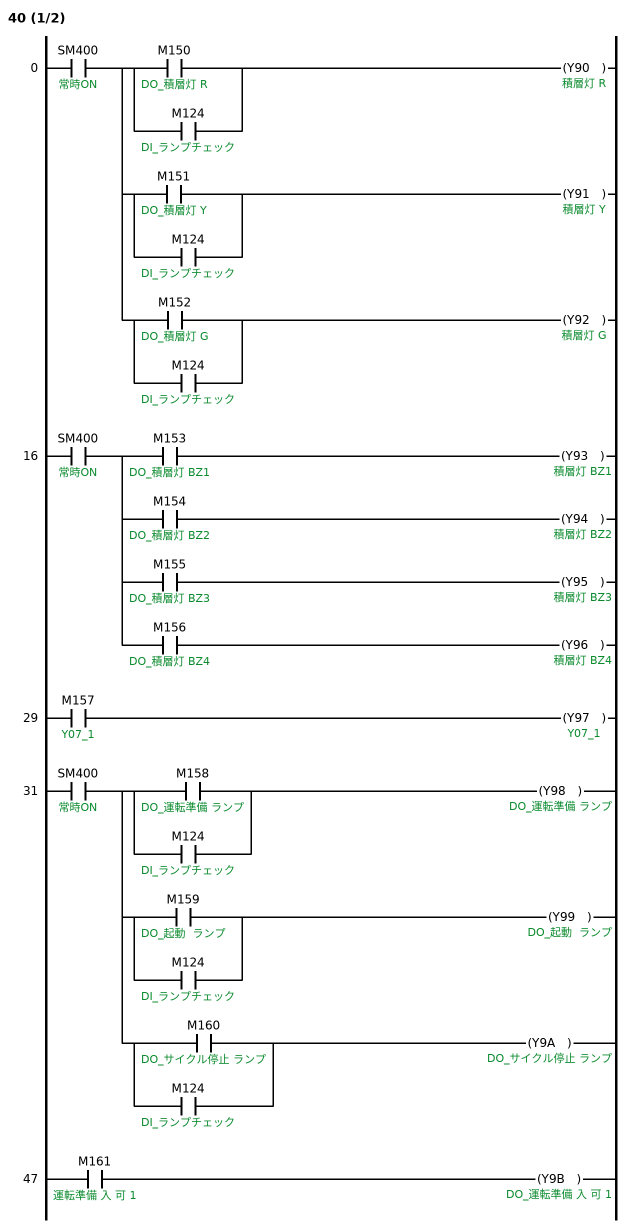
0     LD      SM400  ; 常時ON
      MPS
      LD      M150  ; DO_積層灯 R
      OR      M124  ; DI_ランプチェック
      ANB
      OUT     Y90  ; 積層灯 R
      MRD
      LD      M151  ; DO_積層灯 Y
      OR      M124  ; DI_ランプチェック
      ANB
      OUT     Y91  ; 積層灯 Y
      MPP
      LD      M152  ; DO_積層灯 G
      OR      M124  ; DI_ランプチェック
      ANB
      OUT     Y92  ; 積層灯 G
16    LD      SM400  ; 常時ON
      MPS
      AND     M153  ; DO_積層灯 BZ1
      OUT     Y93  ; 積層灯 BZ1
      MRD
      AND     M154  ; DO_積層灯 BZ2
      OUT     Y94  ; 積層灯 BZ2
      MRD
      AND     M155  ; DO_積層灯 BZ3
      OUT     Y95  ; 積層灯 BZ3
      MPP
      AND     M156  ; DO_積層灯 BZ4
      OUT     Y96  ; 積層灯 BZ4
29    LD      M157  ; Y07_1
      OUT     Y97  ; Y07_1
31    LD      SM400  ; 常時ON
      MPS
      LD      M158  ; DO_運転準備 ランプ
      OR      M124  ; DI_ランプチェック
      ANB
      OUT     Y98  ; DO_運転準備 ランプ
      MRD
      LD      M159  ; DO_起動  ランプ
      OR      M124  ; DI_ランプチェック
      ANB
      OUT     Y99  ; DO_起動  ランプ
      MPP
      LD      M160  ; DO_サイクル停止 ランプ
      OR      M124  ; DI_ランプチェック
      ANB
      OUT     Y9A  ; DO_サイクル停止 ランプ
47    LD      M161  ; 運転準備 入 可 1
      OUT     Y9B  ; DO_運転準備 入 可 1
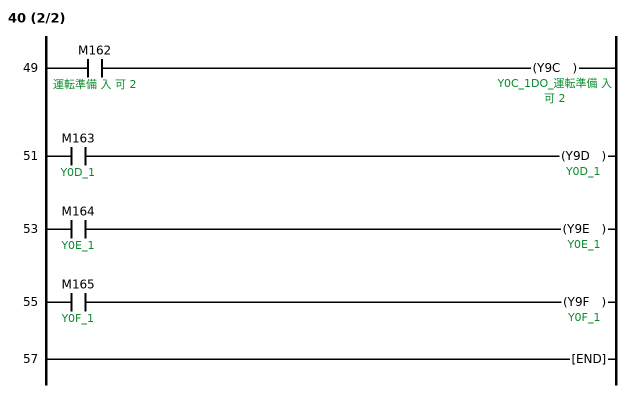
49    LD      M162  ; 運転準備 入 可 2
      OUT     Y9C  ; Y0C_1DO_運転準備 入 可 2
51    LD      M163  ; Y0D_1
      OUT     Y9D  ; Y0D_1
53    LD      M164  ; Y0E_1
      OUT     Y9E  ; Y0E_1
55    LD      M165  ; Y0F_1
      OUT     Y9F  ; Y0F_1
57    END
END_PROGRAM

PROGRAM 42  // スタッカー 出力
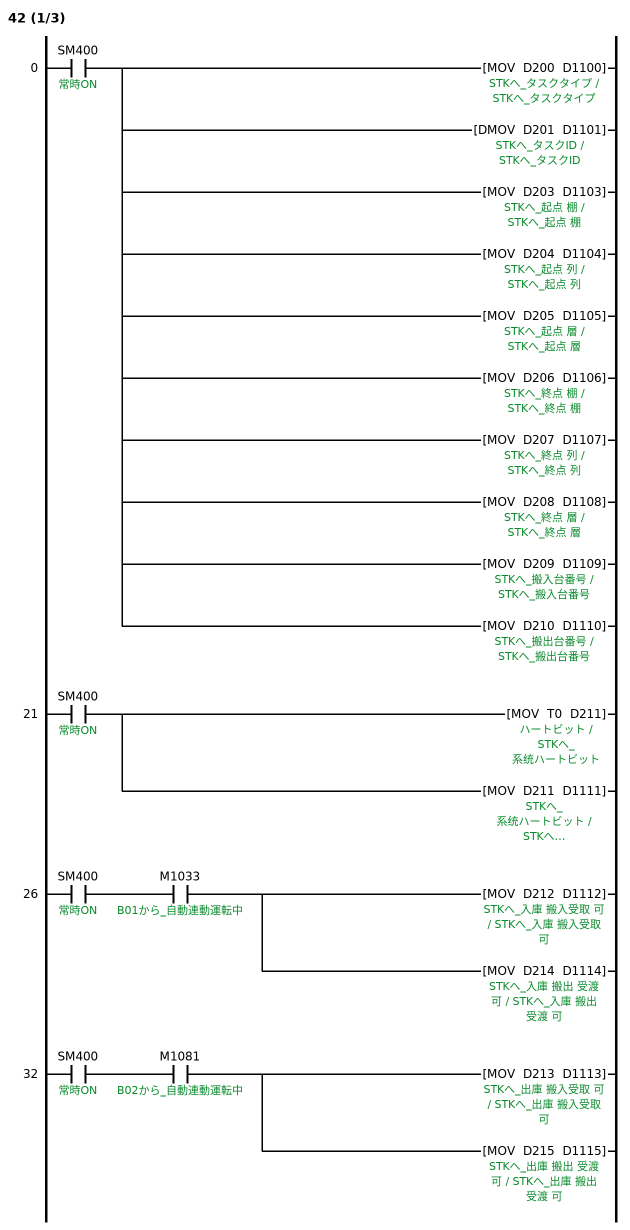
0     LD      SM400  ; 常時ON
      MOV     D200 D1100  ; STKへ_タスクタイプ / STKへ_タスクタイプ
      DMOV    D201 D1101  ; STKへ_タスクID / STKへ_タスクID
      MOV     D203 D1103  ; STKへ_起点 棚 / STKへ_起点 棚
      MOV     D204 D1104  ; STKへ_起点 列 / STKへ_起点 列
      MOV     D205 D1105  ; STKへ_起点 層 / STKへ_起点 層
      MOV     D206 D1106  ; STKへ_終点 棚 / STKへ_終点 棚
      MOV     D207 D1107  ; STKへ_終点 列 / STKへ_終点 列
      MOV     D208 D1108  ; STKへ_終点 層 / STKへ_終点 層
      MOV     D209 D1109  ; STKへ_搬入台番号 / STKへ_搬入台番号
      MOV     D210 D1110  ; STKへ_搬出台番号 / STKへ_搬出台番号
21    LD      SM400  ; 常時ON
      MOV     T0 D211  ; ハートビット / STKへ_系统ハートビット
      MOV     D211 D1111  ; STKへ_系统ハートビット
26    LD      SM400  ; 常時ON
      AND     M1033  ; B01から_自動連動運転中
      MOV     D212 D1112  ; STKへ_入庫 搬入受取 可 / STKへ_入庫 搬入受取 可
      MOV     D214 D1114  ; STKへ_入庫 搬出 受渡 可 / STKへ_入庫 搬出 受渡 可
32    LD      SM400  ; 常時ON
      AND     M1081  ; B02から_自動連動運転中
      MOV     D213 D1113  ; STKへ_出庫 搬入受取 可 / STKへ_出庫 搬入受取 可
      MOV     D215 D1115  ; STKへ_出庫 搬出 受渡 可 / STKへ_出庫 搬出 受渡 可
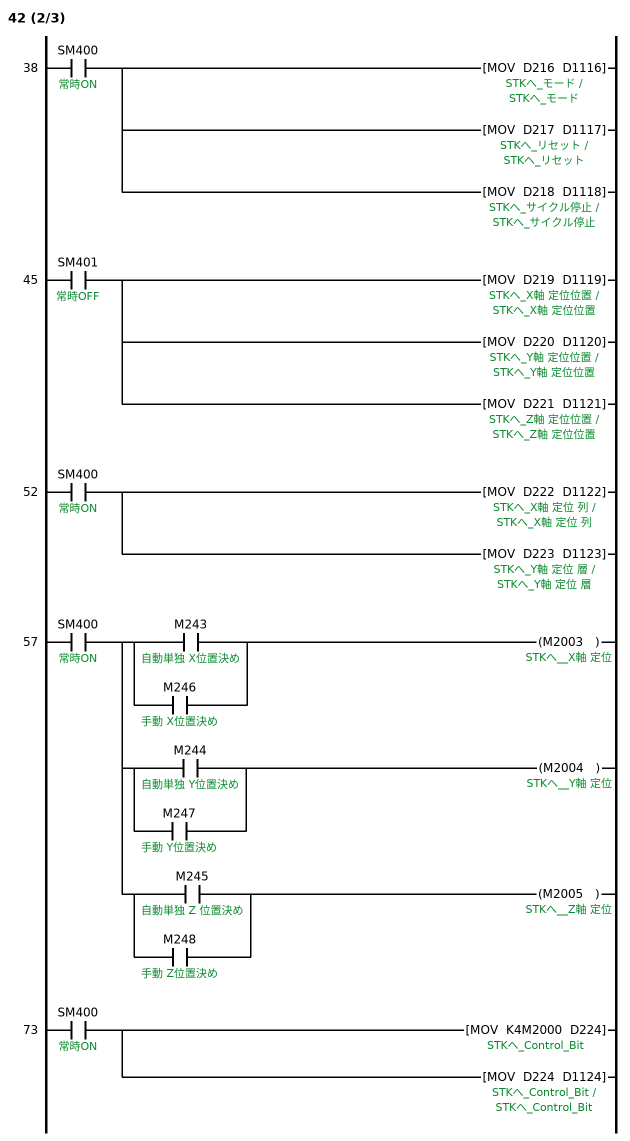
38    LD      SM400  ; 常時ON
      MOV     D216 D1116  ; STKへ_モード / STKへ_モード
      MOV     D217 D1117  ; STKへ_リセット / STKへ_リセット
      MOV     D218 D1118  ; STKへ_サイクル停止 / STKへ_サイクル停止
45    LD      SM401  ; 常時OFF
      MOV     D219 D1119  ; STKへ_X軸 定位位置 / STKへ_X軸 定位位置
      MOV     D220 D1120  ; STKへ_Y軸 定位位置 / STKへ_Y軸 定位位置
      MOV     D221 D1121  ; STKへ_Z軸 定位位置 / STKへ_Z軸 定位位置
52    LD      SM400  ; 常時ON
      MOV     D222 D1122  ; STKへ_X軸 定位 列 / STKへ_X軸 定位 列
      MOV     D223 D1123  ; STKへ_Y軸 定位 層 / STKへ_Y軸 定位 層
57    LD      SM400  ; 常時ON
      MPS
      LD      M243  ; 自動単独 X位置決め
      OR      M246  ; 手動 X位置決め
      ANB
      OUT     M2003  ; STKへ__X軸 定位
      MRD
      LD      M244  ; 自動単独 Y位置決め
      OR      M247  ; 手動 Y位置決め
      ANB
      OUT     M2004  ; STKへ__Y軸 定位
      MPP
      LD      M245  ; 自動単独 Z 位置決め
      OR      M248  ; 手動 Z位置決め
      ANB
      OUT     M2005  ; STKへ__Z軸 定位
73    LD      SM400  ; 常時ON
      MOV     K4M2000 D224  ; STKへ_手動制御リクエスト / STKへ_Control_Bit
      MOV     D224 D1124  ; STKへ_Control_Bit
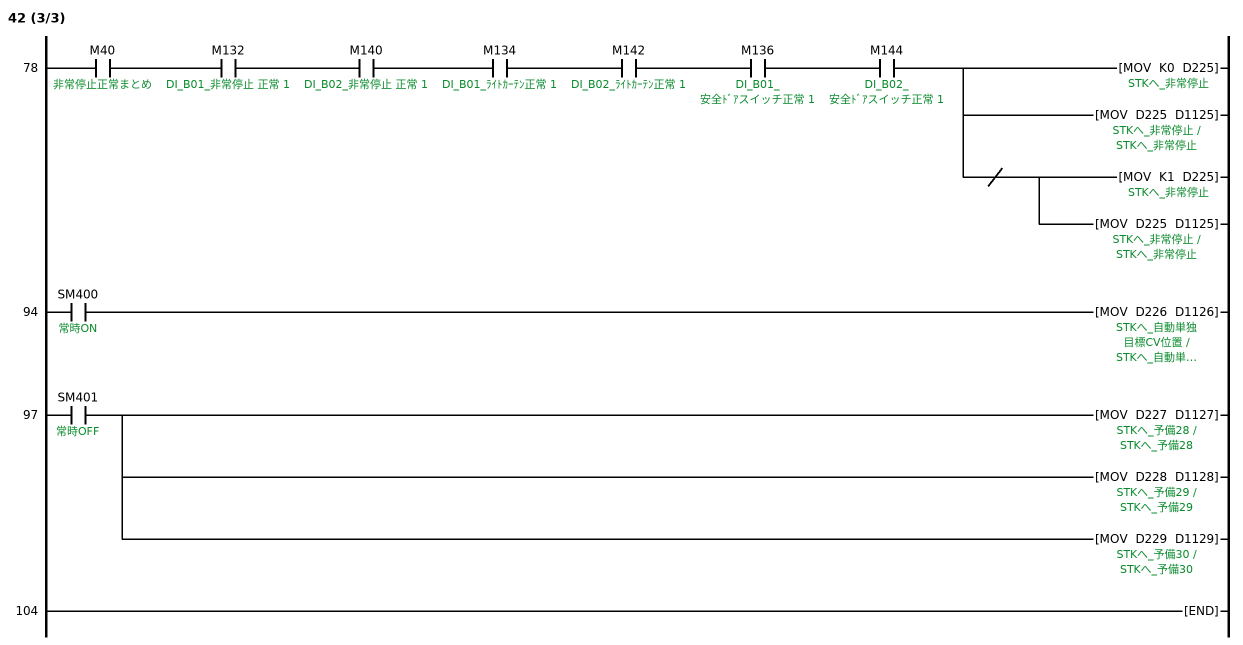
78    LD      M40  ; 非常停止正常まとめ
      AND     M132  ; DI_B01_非常停止 正常 1
      AND     M140  ; DI_B02_非常停止 正常 1
      AND     M134  ; DI_B01_ﾗｲﾄｶｰﾃﾝ正常 1
      AND     M142  ; DI_B02_ﾗｲﾄｶｰﾃﾝ正常 1
      AND     M136  ; DI_B01_安全ﾄﾞｱスイッチ正常 1
      AND     M144  ; DI_B02_安全ﾄﾞｱスイッチ正常 1
      MOV     K0 D225  ; STKへ_非常停止
      MOV     D225 D1125  ; STKへ_非常停止
      INV
      MOV     K1 D225
      MOV     D225 D1125
94    LD      SM400  ; 常時ON
      MOV     D226 D1126  ; STKへ_自動単独 目標CV位置 / STKへ_自動単独 目標CV位置
97    LD      SM401  ; 常時OFF
      MOV     D227 D1127  ; STKへ_予備28 / STKへ_予備28
      MOV     D228 D1128  ; STKへ_予備29 / STKへ_予備29
      MOV     D229 D1129  ; STKへ_予備30 / STKへ_予備30
104   END
END_PROGRAM

PROGRAM 43  // WMS 出力
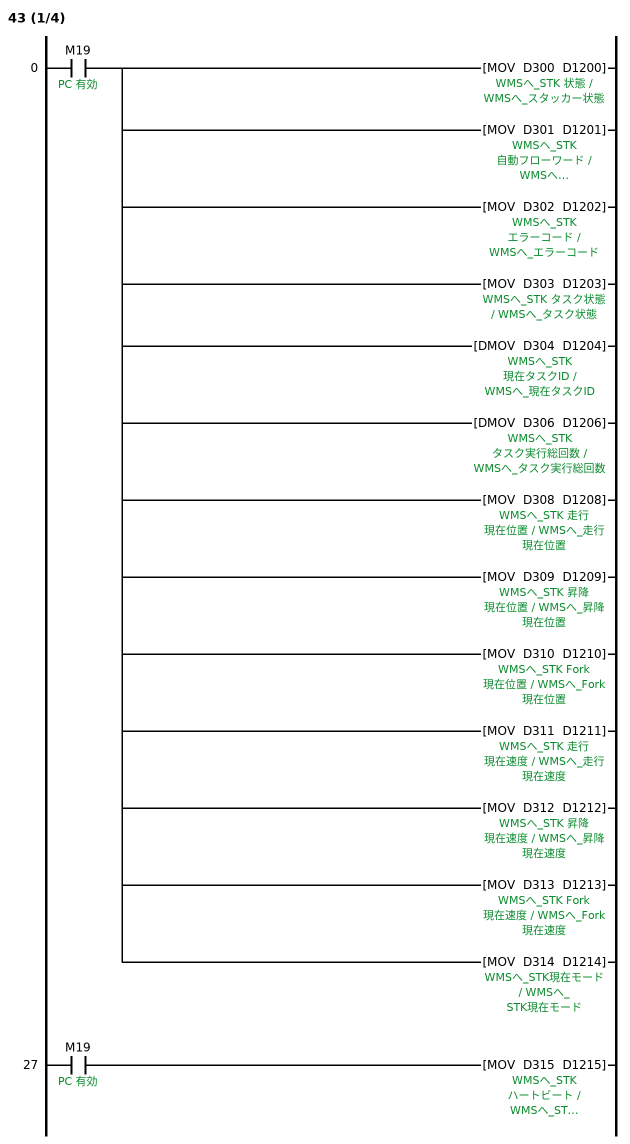
0     LD      M19  ; PC 有効
      MOV     D300 D1200  ; WMSへ_STK 状態 / WMSへ_スタッカー状態
      MOV     D301 D1201  ; WMSへ_STK 自動フローワード / WMSへ_自動フローワード
      MOV     D302 D1202  ; WMSへ_STK エラーコード / WMSへ_エラーコード
      MOV     D303 D1203  ; WMSへ_STK タスク状態 / WMSへ_タスク状態
      DMOV    D304 D1204  ; WMSへ_STK 現在タスクID / WMSへ_現在タスクID
      DMOV    D306 D1206  ; WMSへ_STK タスク実行総回数 / WMSへ_タスク実行総回数
      MOV     D308 D1208  ; WMSへ_STK 走行 現在位置 / WMSへ_走行 現在位置
      MOV     D309 D1209  ; WMSへ_STK 昇降 現在位置 / WMSへ_昇降 現在位置
      MOV     D310 D1210  ; WMSへ_STK Fork 現在位置 / WMSへ_Fork 現在位置
      MOV     D311 D1211  ; WMSへ_STK 走行 現在速度 / WMSへ_走行 現在速度
      MOV     D312 D1212  ; WMSへ_STK 昇降 現在速度 / WMSへ_昇降 現在速度
      MOV     D313 D1213  ; WMSへ_STK Fork 現在速度 / WMSへ_Fork 現在速度
      MOV     D314 D1214  ; WMSへ_STK現在モード / WMSへ_STK現在モード
27    LD      M19  ; PC 有効
      MOV     D315 D1215  ; WMSへ_STK ハートビート / WMSへ_STK ハートビート
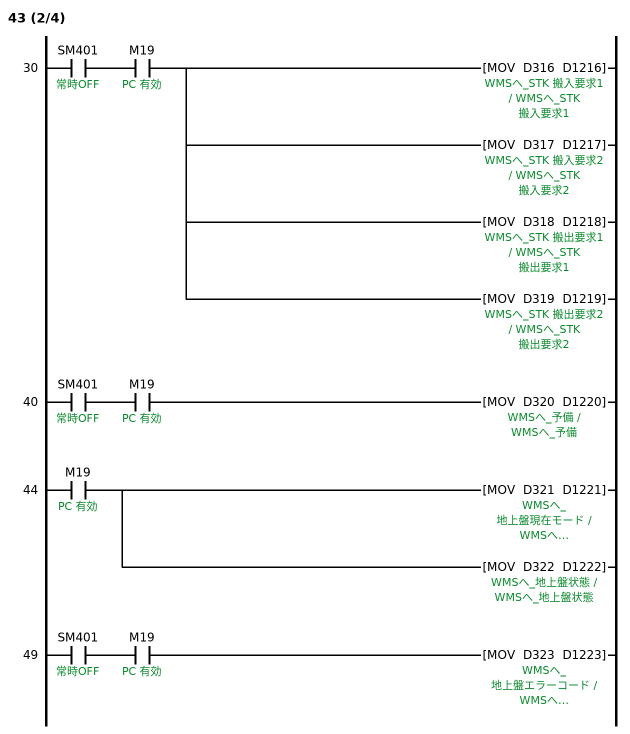
30    LD      SM401  ; 常時OFF
      AND     M19  ; PC 有効
      MOV     D316 D1216  ; WMSへ_STK 搬入要求1 / WMSへ_STK 搬入要求1
      MOV     D317 D1217  ; WMSへ_STK 搬入要求2 / WMSへ_STK 搬入要求2
      MOV     D318 D1218  ; WMSへ_STK 搬出要求1 / WMSへ_STK 搬出要求1
      MOV     D319 D1219  ; WMSへ_STK 搬出要求2 / WMSへ_STK 搬出要求2
40    LD      SM401  ; 常時OFF
      AND     M19  ; PC 有効
      MOV     D320 D1220  ; WMSへ_予備 / WMSへ_予備
44    LD      M19  ; PC 有効
      MOV     D321 D1221  ; WMSへ_地上盤現在モード / WMSへ_地上盤現在モード
      MOV     D322 D1222  ; WMSへ_地上盤状態 / WMSへ_地上盤状態
49    LD      SM401  ; 常時OFF
      AND     M19  ; PC 有効
      MOV     D323 D1223  ; WMSへ_地上盤エラーコード / WMSへ_地上盤エラーコード
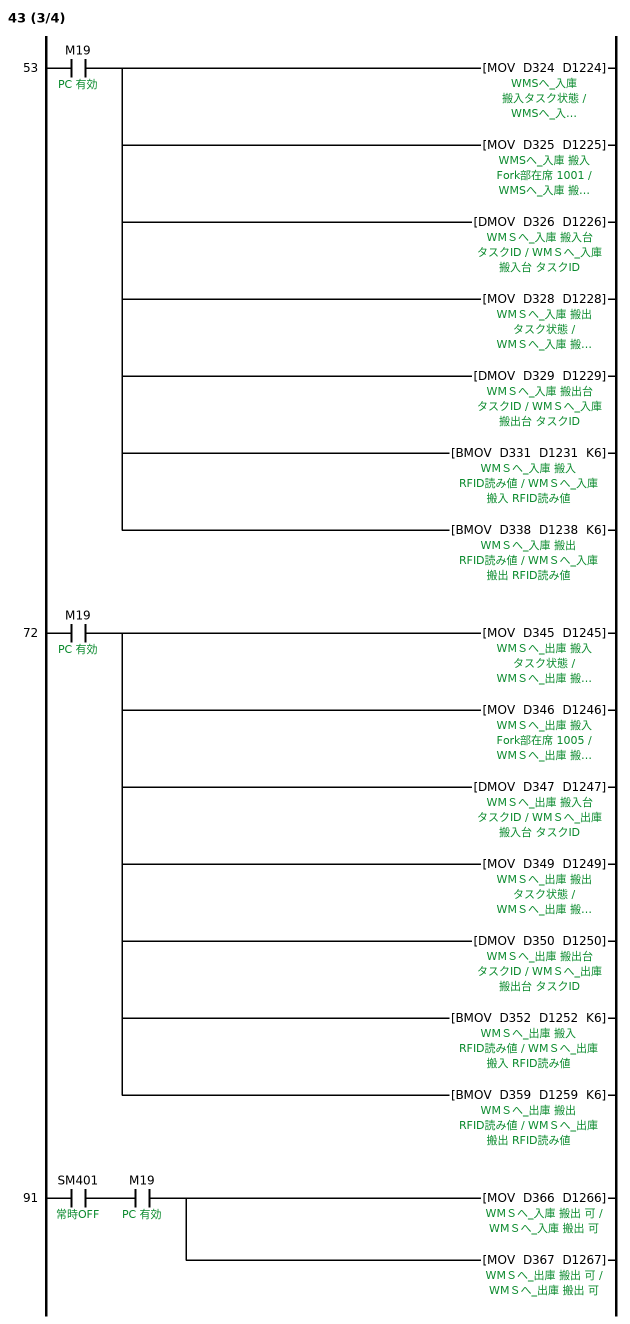
53    LD      M19  ; PC 有効
      MOV     D324 D1224  ; WMSへ_入庫 搬入タスク状態 / WMSへ_入庫 搬入タスク状態
      MOV     D325 D1225  ; WMSへ_入庫 搬入 Fork部在席 1001 / WMSへ_入庫 搬入 Fork在席
      DMOV    D326 D1226  ; WMＳへ_入庫 搬入台 タスクID / WMＳへ_入庫 搬入台 タスクID
      MOV     D328 D1228  ; WMＳへ_入庫 搬出 タスク状態 / WMＳへ_入庫 搬出 タスク状態
      DMOV    D329 D1229  ; WMＳへ_入庫 搬出台 タスクID / WMＳへ_入庫 搬出台 タスクID
      BMOV    D331 D1231 K6  ; WMＳへ_入庫 搬入 RFID読み値 / WMＳへ_入庫 搬入 RFID読み値
      BMOV    D338 D1238 K6  ; WMＳへ_入庫 搬出 RFID読み値 / WMＳへ_入庫 搬出 RFID読み値
72    LD      M19  ; PC 有効
      MOV     D345 D1245  ; WMＳへ_出庫 搬入 タスク状態 / WMＳへ_出庫 搬入 タスク状態
      MOV     D346 D1246  ; WMＳへ_出庫 搬入 Fork部在席 1005 / WMＳへ_出庫 搬入 Fork部在席
      DMOV    D347 D1247  ; WMＳへ_出庫 搬入台 タスクID / WMＳへ_出庫 搬入台 タスクID
      MOV     D349 D1249  ; WMＳへ_出庫 搬出 タスク状態 / WMＳへ_出庫 搬出 タスク状態
      DMOV    D350 D1250  ; WMＳへ_出庫 搬出台 タスクID / WMＳへ_出庫 搬出台 タスクID
      BMOV    D352 D1252 K6  ; WMＳへ_出庫 搬入 RFID読み値 / WMＳへ_出庫 搬入 RFID読み値
      BMOV    D359 D1259 K6  ; WMＳへ_出庫 搬出 RFID読み値 / WMＳへ_出庫 搬出 RFID読み値
91    LD      SM401  ; 常時OFF
      AND     M19  ; PC 有効
      MOV     D366 D1266  ; WMＳへ_入庫 搬出 可 / WMＳへ_入庫 搬出 可
      MOV     D367 D1267  ; WMＳへ_出庫 搬出 可 / WMＳへ_出庫 搬出 可
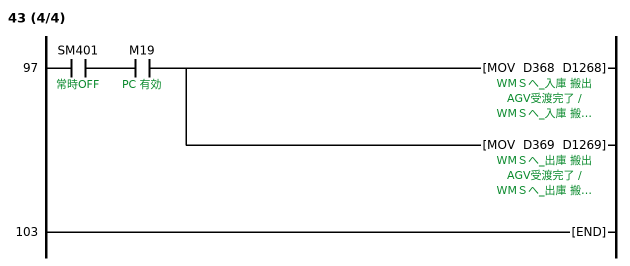
97    LD      SM401  ; 常時OFF
      AND     M19  ; PC 有効
      MOV     D368 D1268  ; WMＳへ_入庫 搬出 AGV受渡完了 / WMＳへ_入庫 搬出 AGV受渡完了
      MOV     D369 D1269  ; WMＳへ_出庫 搬出 AGV受渡完了 / WMＳへ_出庫 搬出 AGV受渡完了
103   END
END_PROGRAM

FUNCTION_BLOCK I+ST_02f34114d45741f9
VAR_INPUT
  __IST_EN_IN : BOOL;
END_VAR
VAR_OUTPUT
  __IST_EN_OUT : BOOL;
END_VAR
(* IST HEADER START *)
IF NOT __IST_EN_IN THEN __IST_EN_OUT:=FALSE; RETURN; END_IF;
(* VERSION=1:TYPE=STB *)
(* IST HEADER END *)
Z0:=(Alone.起点列 - 1) * 5 + (Alone.起点層 - 1); (*起点位置*)
END_FUNCTION_BLOCK

FUNCTION_BLOCK I+ST_08ba2391820a4452
VAR_INPUT
  __IST_EN_IN : BOOL;
END_VAR
VAR_OUTPUT
  __IST_EN_OUT : BOOL;
END_VAR
(* IST HEADER START *)
IF NOT __IST_EN_IN THEN __IST_EN_OUT:=FALSE; RETURN; END_IF;
(* VERSION=1:TYPE=STB *)
(* IST HEADER END *)
Z1:=(Alone.終点列 - 1) * 5 + (Alone.終点層 - 1); (*目的位置*)
END_FUNCTION_BLOCK

PROGRAM 13  // STK 自動/単独ﾓｰﾄﾞ
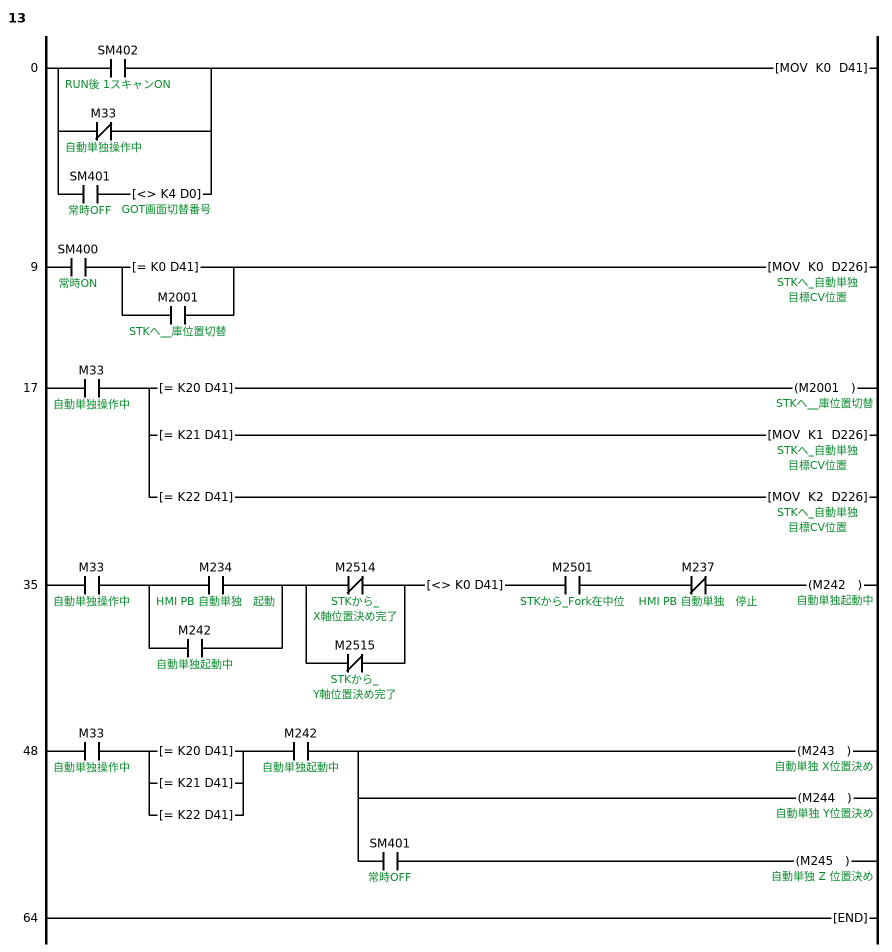
0     LD      SM402  ; RUN後 1スキャンON
      ORI     M33  ; 自動単独操作中
      LD      SM401  ; 常時OFF
      AND<>   K4 D0  ; GOT画面切替番号
      ORB
      MOV     K0 D41
9     LD      SM400  ; 常時ON
      LD=     K0 D41
      OR      M2001  ; STKへ__庫位置切替
      ANB
      MOV     K0 D226  ; STKへ_自動単独 目標CV位置
17    LD      M33  ; 自動単独操作中
      MPS
      AND=    K20 D41
      OUT     M2001  ; STKへ__庫位置切替
      MRD
      AND=    K21 D41
      MOV     K1 D226
      MPP
      AND=    K22 D41
      MOV     K2 D226
35    LD      M33  ; 自動単独操作中
      LD      M234  ; HMI PB 自動単独　起動
      OR      M242  ; 自動単独起動中
      ANB
      LDI     M2514  ; STKから_X軸位置決め完了
      ORI     M2515  ; STKから_Y軸位置決め完了
      ANB
      AND<>   K0 D41
      AND     M2501  ; STKから_Fork在中位
      ANI     M237  ; HMI PB 自動単独　停止
      OUT     M242  ; 自動単独起動中
48    LD      M33  ; 自動単独操作中
      LD=     K20 D41
      OR=     K21 D41
      OR=     K22 D41
      ANB
      AND     M242  ; 自動単独起動中
      OUT     M243  ; 自動単独 X位置決め
      OUT     M244  ; 自動単独 Y位置決め
      AND     SM401  ; 常時OFF
      OUT     M245  ; 自動単独 Z 位置決め
64    END
END_PROGRAM

PROGRAM 04  // B01 CC-LinkIE XYD 入力
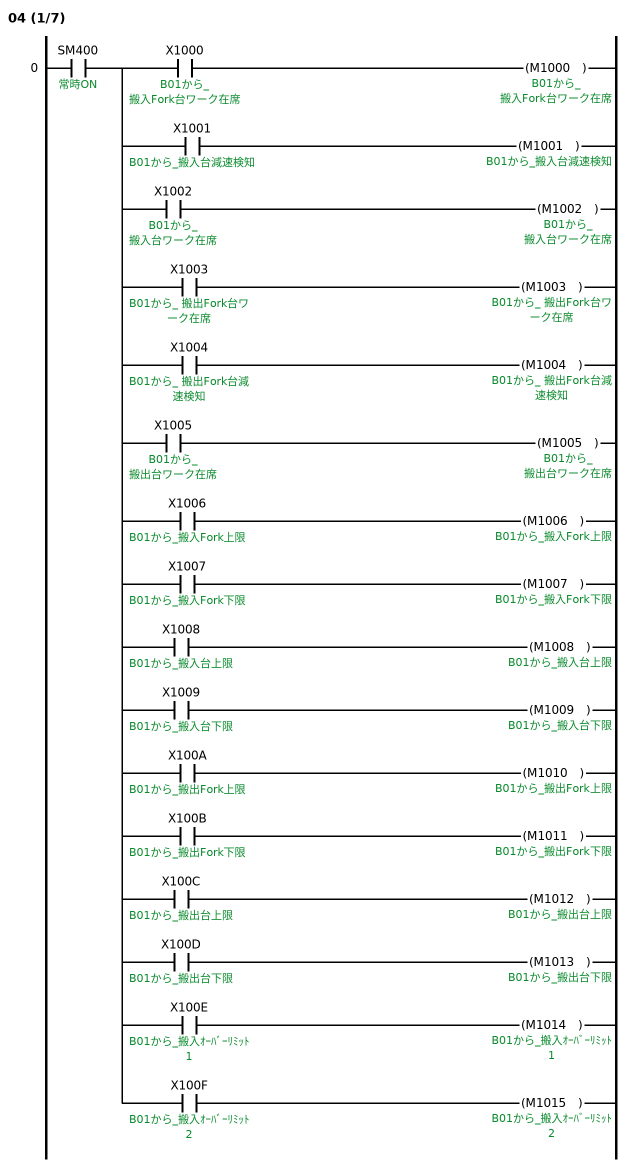
0     LD      SM400  ; 常時ON
      MPS
      AND     X1000  ; B01から_搬入Fork台ワーク在席
      OUT     M1000  ; B01から_搬入Fork台ワーク在席
      MRD
      AND     X1001  ; B01から_搬入台減速検知
      OUT     M1001  ; B01から_搬入台減速検知
      MRD
      AND     X1002  ; B01から_搬入台ワーク在席
      OUT     M1002  ; B01から_搬入台ワーク在席
      MRD
      AND     X1003  ; B01から_ 搬出Fork台ワーク在席
      OUT     M1003  ; B01から_ 搬出Fork台ワーク在席
      MRD
      AND     X1004  ; B01から_ 搬出Fork台減速検知
      OUT     M1004  ; B01から_ 搬出Fork台減速検知
      MRD
      AND     X1005  ; B01から_ 搬出台ワーク在席
      OUT     M1005  ; B01から_ 搬出台ワーク在席
      MRD
      AND     X1006  ; B01から_搬入Fork上限
      OUT     M1006  ; B01から_搬入Fork上限
      MRD
      AND     X1007  ; B01から_搬入Fork下限
      OUT     M1007  ; B01から_搬入Fork下限
      MRD
      AND     X1008  ; B01から_搬入台上限
      OUT     M1008  ; B01から_搬入台上限
      MRD
      AND     X1009  ; B01から_搬入台下限
      OUT     M1009  ; B01から_搬入台下限
      MRD
      AND     X100A  ; B01から_搬出Fork上限
      OUT     M1010  ; B01から_搬出Fork上限
      MRD
      AND     X100B  ; B01から_搬出Fork下限
      OUT     M1011  ; B01から_搬出Fork下限
      MRD
      AND     X100C  ; B01から_搬出台上限
      OUT     M1012  ; B01から_搬出台上限
      MRD
      AND     X100D  ; B01から_搬出台下限
      OUT     M1013  ; B01から_搬出台下限
      MRD
      AND     X100E  ; B01から_搬入ｵｰﾊﾞｰﾘﾐｯﾄ 1
      OUT     M1014  ; B01から_搬入ｵｰﾊﾞｰﾘﾐｯﾄ 1
      MPP
      AND     X100F  ; B01から_搬入ｵｰﾊﾞｰﾘﾐｯﾄ 2
      OUT     M1015  ; B01から_搬入ｵｰﾊﾞｰﾘﾐｯﾄ 2
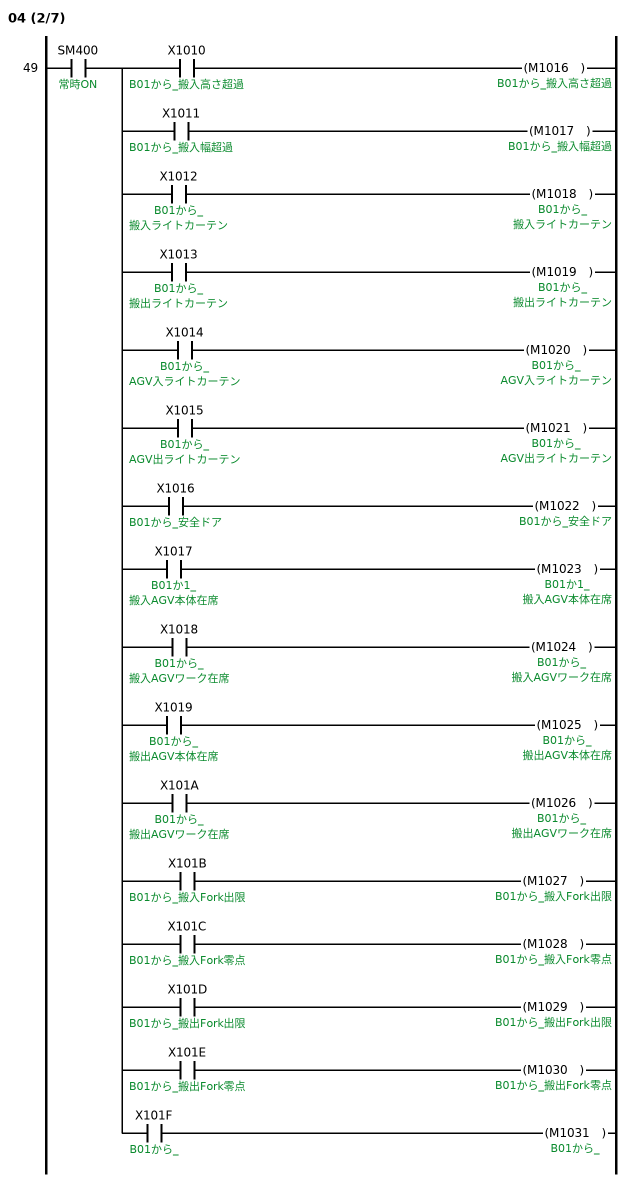
49    LD      SM400  ; 常時ON
      MPS
      AND     X1010  ; B01から_搬入高さ超過
      OUT     M1016  ; B01から_搬入高さ超過
      MRD
      AND     X1011  ; B01から_搬入幅超過
      OUT     M1017  ; B01から_搬入幅超過
      MRD
      AND     X1012  ; B01から_搬入ライトカーテン
      OUT     M1018  ; B01から_搬入ライトカーテン
      MRD
      AND     X1013  ; B01から_搬出ライトカーテン
      OUT     M1019  ; B01から_搬出ライトカーテン
      MRD
      AND     X1014  ; B01から_AGV入ライトカーテン
      OUT     M1020  ; B01から_AGV入ライトカーテン
      MRD
      AND     X1015  ; B01から_AGV出ライトカーテン
      OUT     M1021  ; B01から_AGV出ライトカーテン
      MRD
      AND     X1016  ; B01から_安全ドア
      OUT     M1022  ; B01から_安全ドア
      MRD
      AND     X1017  ; B01か1_搬入AGV本体在席
      OUT     M1023  ; B01か1_搬入AGV本体在席
      MRD
      AND     X1018  ; B01から_搬入AGVワーク在席
      OUT     M1024  ; B01から_搬入AGVワーク在席
      MRD
      AND     X1019  ; B01から_搬出AGV本体在席
      OUT     M1025  ; B01から_搬出AGV本体在席
      MRD
      AND     X101A  ; B01から_搬出AGVワーク在席
      OUT     M1026  ; B01から_搬出AGVワーク在席
      MRD
      AND     X101B  ; B01から_搬入Fork出限
      OUT     M1027  ; B01から_搬入Fork出限
      MRD
      AND     X101C  ; B01から_搬入Fork零点
      OUT     M1028  ; B01から_搬入Fork零点
      MRD
      AND     X101D  ; B01から_搬出Fork出限
      OUT     M1029  ; B01から_搬出Fork出限
      MRD
      AND     X101E  ; B01から_搬出Fork零点
      OUT     M1030  ; B01から_搬出Fork零点
      MPP
      AND     X101F  ; B01から_
      OUT     M1031  ; B01から_
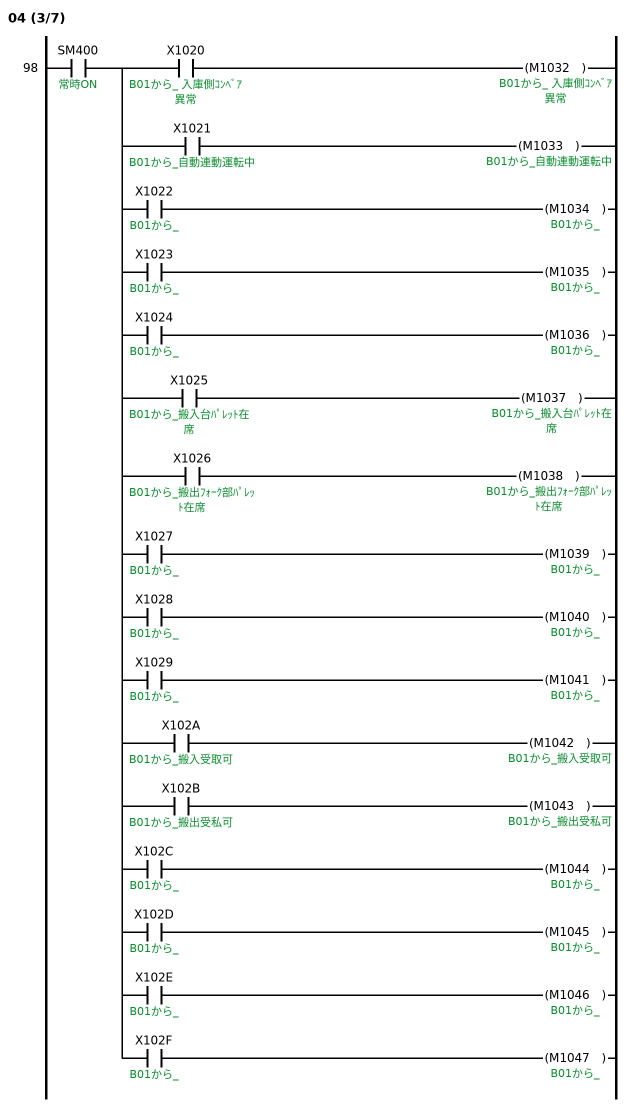
98    LD      SM400  ; 常時ON
      MPS
      AND     X1020  ; B01から_ 入庫側ｺﾝﾍﾞｱ 異常
      OUT     M1032  ; B01から_ 入庫側ｺﾝﾍﾞｱ 異常
      MRD
      AND     X1021  ; B01から_自動連動運転中
      OUT     M1033  ; B01から_自動連動運転中
      MRD
      AND     X1022  ; B01から_
      OUT     M1034  ; B01から_
      MRD
      AND     X1023  ; B01から_
      OUT     M1035  ; B01から_
      MRD
      AND     X1024  ; B01から_
      OUT     M1036  ; B01から_
      MRD
      AND     X1025  ; B01から_搬入台ﾊﾟﾚｯﾄ在席
      OUT     M1037  ; B01から_搬入台ﾊﾟﾚｯﾄ在席
      MRD
      AND     X1026  ; B01から_搬出ﾌｫｰｸ部ﾊﾟﾚｯﾄ在席
      OUT     M1038  ; B01から_搬出ﾌｫｰｸ部ﾊﾟﾚｯﾄ在席
      MRD
      AND     X1027  ; B01から_
      OUT     M1039  ; B01から_
      MRD
      AND     X1028  ; B01から_
      OUT     M1040  ; B01から_
      MRD
      AND     X1029  ; B01から_
      OUT     M1041  ; B01から_
      MRD
      AND     X102A  ; B01から_搬入受取可
      OUT     M1042  ; B01から_搬入受取可
      MRD
      AND     X102B  ; B01から_搬出受私可
      OUT     M1043  ; B01から_搬出受私可
      MRD
      AND     X102C  ; B01から_
      OUT     M1044  ; B01から_
      MRD
      AND     X102D  ; B01から_
      OUT     M1045  ; B01から_
      MRD
      AND     X102E  ; B01から_
      OUT     M1046  ; B01から_
      MPP
      AND     X102F  ; B01から_
      OUT     M1047  ; B01から_
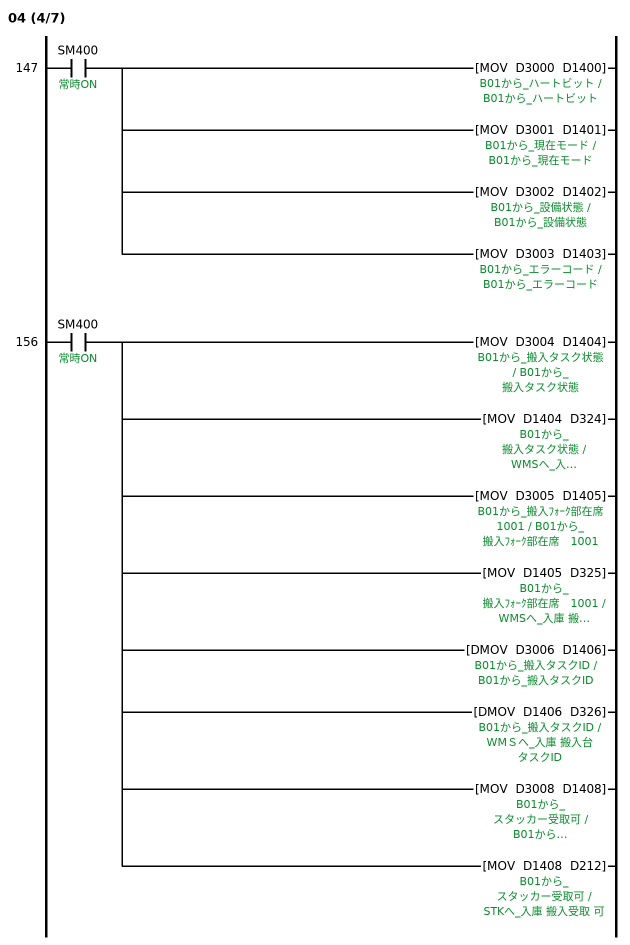
147   LD      SM400  ; 常時ON
      MOV     D3000 D1400  ; B01から_ハートビット / B01から_ハートビット
      MOV     D3001 D1401  ; B01から_現在モード / B01から_現在モード
      MOV     D3002 D1402  ; B01から_設備状態 / B01から_設備状態
      MOV     D3003 D1403  ; B01から_エラーコード / B01から_エラーコード
156   LD      SM400  ; 常時ON
      MOV     D3004 D1404  ; B01から_搬入タスク状態 / B01から_搬入タスク状態
      MOV     D1404 D324  ; WMSへ_入庫 搬入タスク状態
      MOV     D3005 D1405  ; B01から_搬入ﾌｫｰｸ部在席　1001 / B01から_搬入ﾌｫｰｸ部在席　1001
      MOV     D1405 D325  ; WMSへ_入庫 搬入 Fork部在席 1001
      DMOV    D3006 D1406  ; B01から_搬入タスクID / B01から_搬入タスクID
      DMOV    D1406 D326  ; WMＳへ_入庫 搬入台 タスクID
      MOV     D3008 D1408  ; B01から_スタッカー受取可 / B01から_スタッカー受取可
      MOV     D1408 D212  ; STKへ_入庫 搬入受取 可
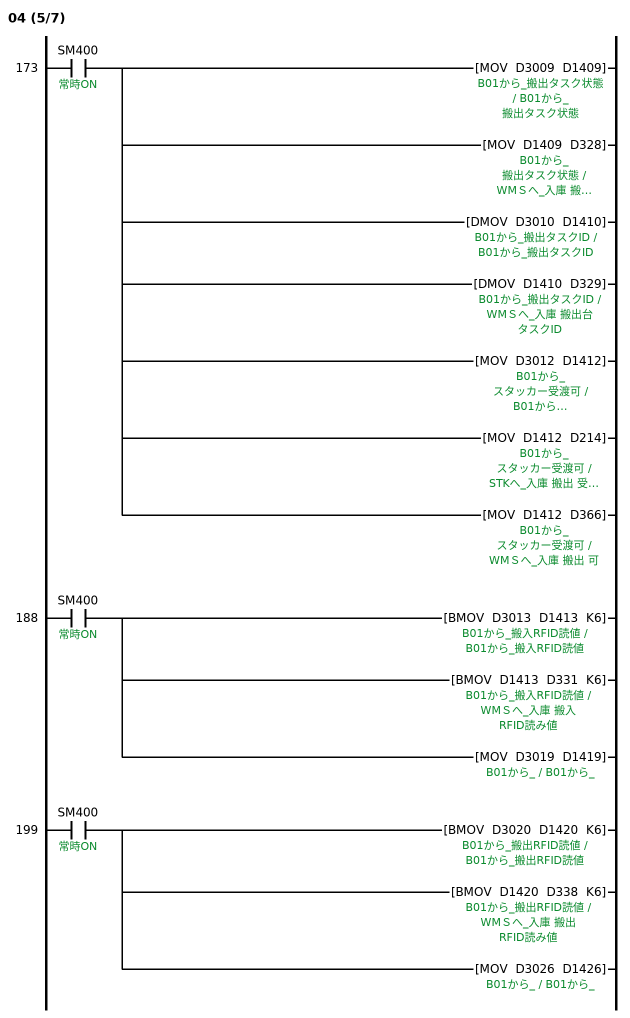
173   LD      SM400  ; 常時ON
      MOV     D3009 D1409  ; B01から_搬出タスク状態 / B01から_搬出タスク状態
      MOV     D1409 D328  ; WMＳへ_入庫 搬出 タスク状態
      DMOV    D3010 D1410  ; B01から_搬出タスクID / B01から_搬出タスクID
      DMOV    D1410 D329  ; WMＳへ_入庫 搬出台 タスクID
      MOV     D3012 D1412  ; B01から_スタッカー受渡可 / B01から_スタッカー受渡可
      MOV     D1412 D214  ; STKへ_入庫 搬出 受渡 可
      MOV     D1412 D366  ; WMＳへ_入庫 搬出 可
188   LD      SM400  ; 常時ON
      BMOV    D3013 D1413 K6  ; B01から_搬入RFID読値 / B01から_搬入RFID読値
      BMOV    D1413 D331 K6  ; WMＳへ_入庫 搬入 RFID読み値
      MOV     D3019 D1419  ; B01から_ / B01から_
199   LD      SM400  ; 常時ON
      BMOV    D3020 D1420 K6  ; B01から_搬出RFID読値 / B01から_搬出RFID読値
      BMOV    D1420 D338 K6  ; WMＳへ_入庫 搬出 RFID読み値
      MOV     D3026 D1426  ; B01から_ / B01から_
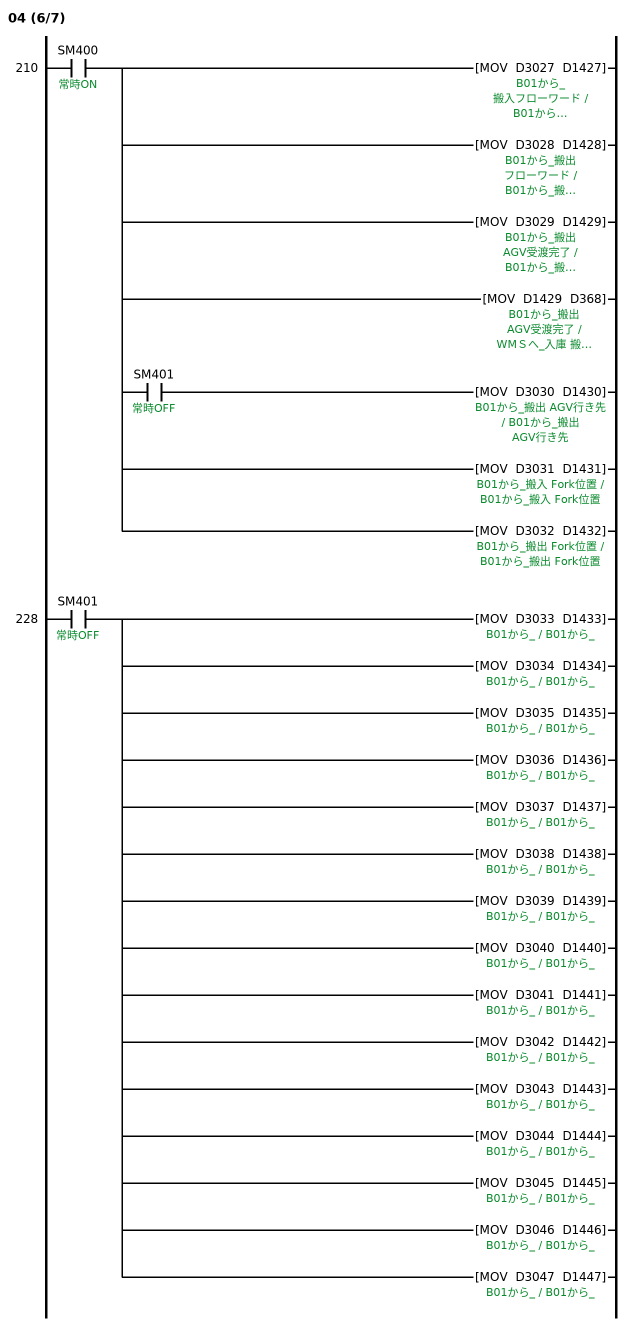
210   LD      SM400  ; 常時ON
      MOV     D3027 D1427  ; B01から_搬入フローワード / B01から_搬入フローワード
      MOV     D3028 D1428  ; B01から_搬出 フローワード / B01から_搬出 フローワード
      MOV     D3029 D1429  ; B01から_搬出 AGV受渡完了 / B01から_搬出 AGV受渡完了
      MOV     D1429 D368  ; WMＳへ_入庫 搬出 AGV受渡完了
      MPS
      AND     SM401  ; 常時OFF
      MOV     D3030 D1430  ; B01から_搬出 AGV行き先 / B01から_搬出 AGV行き先
      MPP
      MOV     D3031 D1431  ; B01から_搬入 Fork位置 / B01から_搬入 Fork位置
      MOV     D3032 D1432  ; B01から_搬出 Fork位置 / B01から_搬出 Fork位置
228   LD      SM401  ; 常時OFF
      MOV     D3033 D1433  ; B01から_ / B01から_
      MOV     D3034 D1434  ; B01から_ / B01から_
      MOV     D3035 D1435  ; B01から_ / B01から_
      MOV     D3036 D1436  ; B01から_ / B01から_
      MOV     D3037 D1437  ; B01から_ / B01から_
      MOV     D3038 D1438  ; B01から_ / B01から_
      MOV     D3039 D1439  ; B01から_ / B01から_
      MOV     D3040 D1440  ; B01から_ / B01から_
      MOV     D3041 D1441  ; B01から_ / B01から_
      MOV     D3042 D1442  ; B01から_ / B01から_
      MOV     D3043 D1443  ; B01から_ / B01から_
      MOV     D3044 D1444  ; B01から_ / B01から_
      MOV     D3045 D1445  ; B01から_ / B01から_
      MOV     D3046 D1446  ; B01から_ / B01から_
      MOV     D3047 D1447  ; B01から_ / B01から_
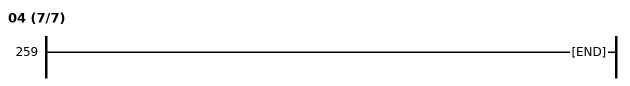
259   END
END_PROGRAM

PROGRAM 44  // B01 CC-LinkIE XVD 出力
0     END
END_PROGRAM

PROGRAM 05  // B02 CC-LinkIE XYD 入力
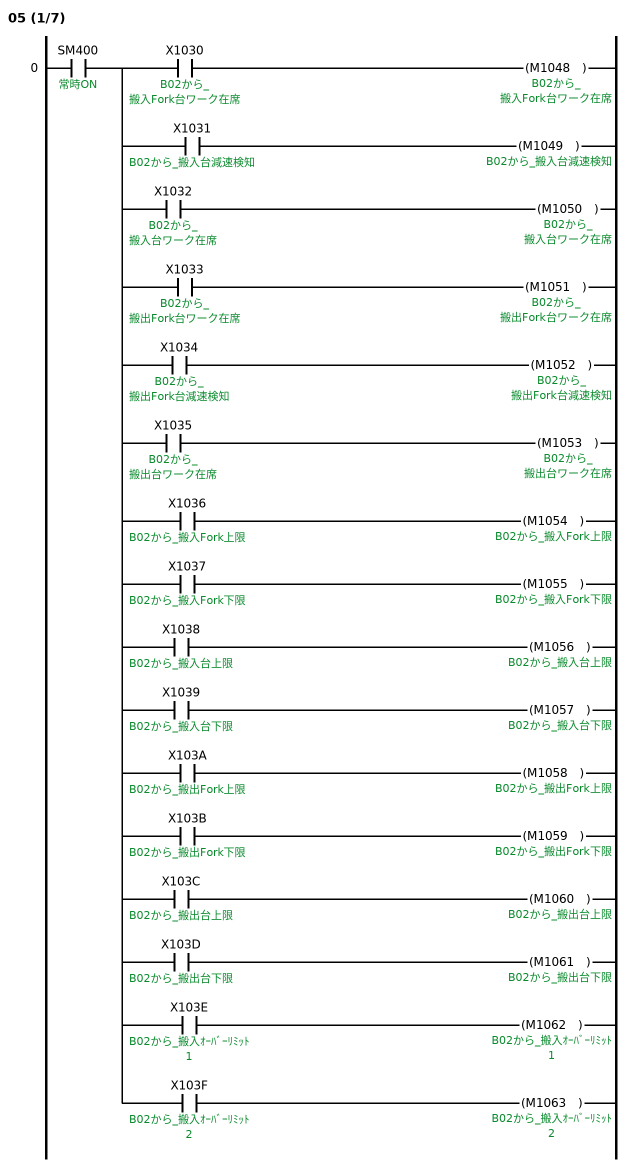
0     LD      SM400  ; 常時ON
      MPS
      AND     X1030  ; B02から_搬入Fork台ワーク在席
      OUT     M1048  ; B02から_搬入Fork台ワーク在席
      MRD
      AND     X1031  ; B02から_搬入台減速検知
      OUT     M1049  ; B02から_搬入台減速検知
      MRD
      AND     X1032  ; B02から_搬入台ワーク在席
      OUT     M1050  ; B02から_搬入台ワーク在席
      MRD
      AND     X1033  ; B02から_搬出Fork台ワーク在席
      OUT     M1051  ; B02から_搬出Fork台ワーク在席
      MRD
      AND     X1034  ; B02から_搬出Fork台減速検知
      OUT     M1052  ; B02から_搬出Fork台減速検知
      MRD
      AND     X1035  ; B02から_搬出台ワーク在席
      OUT     M1053  ; B02から_搬出台ワーク在席
      MRD
      AND     X1036  ; B02から_搬入Fork上限
      OUT     M1054  ; B02から_搬入Fork上限
      MRD
      AND     X1037  ; B02から_搬入Fork下限
      OUT     M1055  ; B02から_搬入Fork下限
      MRD
      AND     X1038  ; B02から_搬入台上限
      OUT     M1056  ; B02から_搬入台上限
      MRD
      AND     X1039  ; B02から_搬入台下限
      OUT     M1057  ; B02から_搬入台下限
      MRD
      AND     X103A  ; B02から_搬出Fork上限
      OUT     M1058  ; B02から_搬出Fork上限
      MRD
      AND     X103B  ; B02から_搬出Fork下限
      OUT     M1059  ; B02から_搬出Fork下限
      MRD
      AND     X103C  ; B02から_搬出台上限
      OUT     M1060  ; B02から_搬出台上限
      MRD
      AND     X103D  ; B02から_搬出台下限
      OUT     M1061  ; B02から_搬出台下限
      MRD
      AND     X103E  ; B02から_搬入ｵｰﾊﾞｰﾘﾐｯﾄ 1
      OUT     M1062  ; B02から_搬入ｵｰﾊﾞｰﾘﾐｯﾄ 1
      MPP
      AND     X103F  ; B02から_搬入ｵｰﾊﾞｰﾘﾐｯﾄ 2
      OUT     M1063  ; B02から_搬入ｵｰﾊﾞｰﾘﾐｯﾄ 2
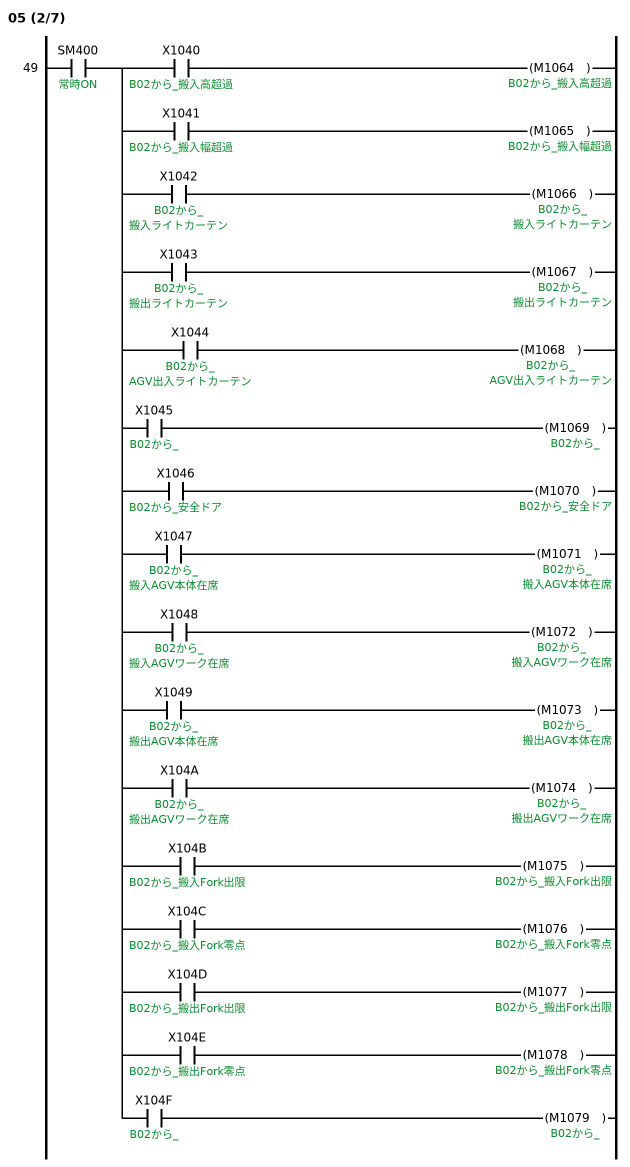
49    LD      SM400  ; 常時ON
      MPS
      AND     X1040  ; B02から_搬入高超過
      OUT     M1064  ; B02から_搬入高超過
      MRD
      AND     X1041  ; B02から_搬入幅超過
      OUT     M1065  ; B02から_搬入幅超過
      MRD
      AND     X1042  ; B02から_搬入ライトカーテン
      OUT     M1066  ; B02から_搬入ライトカーテン
      MRD
      AND     X1043  ; B02から_搬出ライトカーテン
      OUT     M1067  ; B02から_搬出ライトカーテン
      MRD
      AND     X1044  ; B02から_AGV出入ライトカーテン
      OUT     M1068  ; B02から_AGV出入ライトカーテン
      MRD
      AND     X1045  ; B02から_
      OUT     M1069  ; B02から_
      MRD
      AND     X1046  ; B02から_安全ドア
      OUT     M1070  ; B02から_安全ドア
      MRD
      AND     X1047  ; B02から_搬入AGV本体在席
      OUT     M1071  ; B02から_搬入AGV本体在席
      MRD
      AND     X1048  ; B02から_搬入AGVワーク在席
      OUT     M1072  ; B02から_搬入AGVワーク在席
      MRD
      AND     X1049  ; B02から_搬出AGV本体在席
      OUT     M1073  ; B02から_搬出AGV本体在席
      MRD
      AND     X104A  ; B02から_搬出AGVワーク在席
      OUT     M1074  ; B02から_搬出AGVワーク在席
      MRD
      AND     X104B  ; B02から_搬入Fork出限
      OUT     M1075  ; B02から_搬入Fork出限
      MRD
      AND     X104C  ; B02から_搬入Fork零点
      OUT     M1076  ; B02から_搬入Fork零点
      MRD
      AND     X104D  ; B02から_搬出Fork出限
      OUT     M1077  ; B02から_搬出Fork出限
      MRD
      AND     X104E  ; B02から_搬出Fork零点
      OUT     M1078  ; B02から_搬出Fork零点
      MPP
      AND     X104F  ; B02から_
      OUT     M1079  ; B02から_
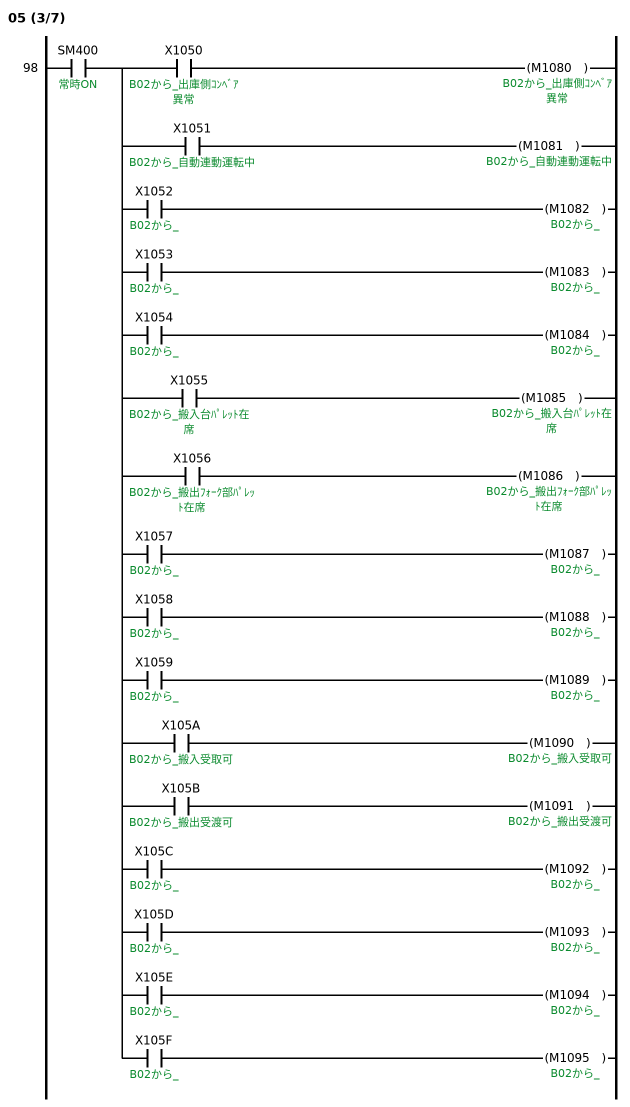
98    LD      SM400  ; 常時ON
      MPS
      AND     X1050  ; B02から_出庫側ｺﾝﾍﾞｱ 異常
      OUT     M1080  ; B02から_出庫側ｺﾝﾍﾞｱ 異常
      MRD
      AND     X1051  ; B02から_自動連動運転中
      OUT     M1081  ; B02から_自動連動運転中
      MRD
      AND     X1052  ; B02から_
      OUT     M1082  ; B02から_
      MRD
      AND     X1053  ; B02から_
      OUT     M1083  ; B02から_
      MRD
      AND     X1054  ; B02から_
      OUT     M1084  ; B02から_
      MRD
      AND     X1055  ; B02から_搬入台ﾊﾟﾚｯﾄ在席
      OUT     M1085  ; B02から_搬入台ﾊﾟﾚｯﾄ在席
      MRD
      AND     X1056  ; B02から_搬出ﾌｫｰｸ部ﾊﾟﾚｯﾄ在席
      OUT     M1086  ; B02から_搬出ﾌｫｰｸ部ﾊﾟﾚｯﾄ在席
      MRD
      AND     X1057  ; B02から_
      OUT     M1087  ; B02から_
      MRD
      AND     X1058  ; B02から_
      OUT     M1088  ; B02から_
      MRD
      AND     X1059  ; B02から_
      OUT     M1089  ; B02から_
      MRD
      AND     X105A  ; B02から_搬入受取可
      OUT     M1090  ; B02から_搬入受取可
      MRD
      AND     X105B  ; B02から_搬出受渡可
      OUT     M1091  ; B02から_搬出受渡可
      MRD
      AND     X105C  ; B02から_
      OUT     M1092  ; B02から_
      MRD
      AND     X105D  ; B02から_
      OUT     M1093  ; B02から_
      MRD
      AND     X105E  ; B02から_
      OUT     M1094  ; B02から_
      MPP
      AND     X105F  ; B02から_
      OUT     M1095  ; B02から_
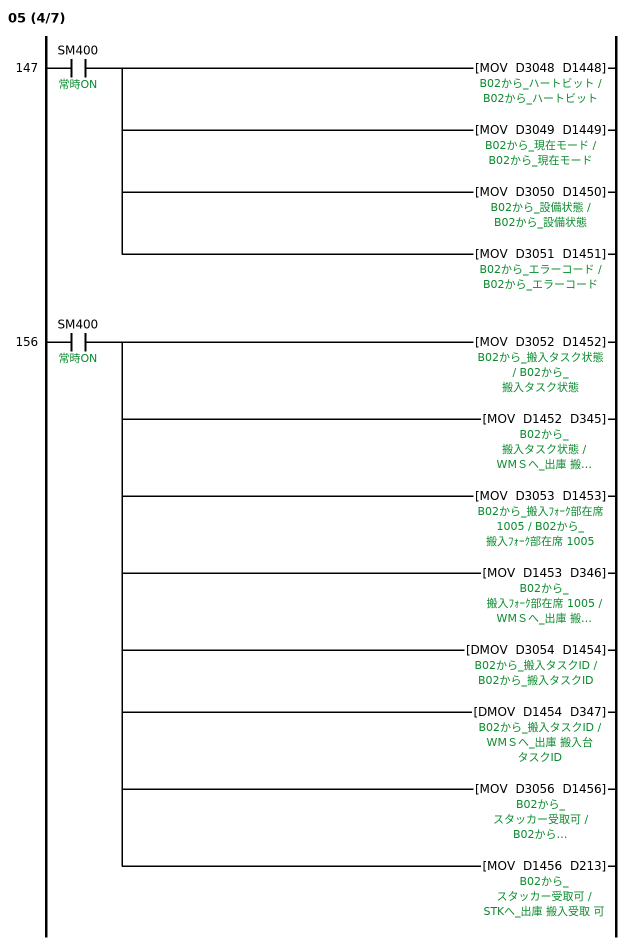
147   LD      SM400  ; 常時ON
      MOV     D3048 D1448  ; B02から_ハートビット / B02から_ハートビット
      MOV     D3049 D1449  ; B02から_現在モード / B02から_現在モード
      MOV     D3050 D1450  ; B02から_設備状態 / B02から_設備状態
      MOV     D3051 D1451  ; B02から_エラーコード / B02から_エラーコード
156   LD      SM400  ; 常時ON
      MOV     D3052 D1452  ; B02から_搬入タスク状態 / B02から_搬入タスク状態
      MOV     D1452 D345  ; WMＳへ_出庫 搬入 タスク状態
      MOV     D3053 D1453  ; B02から_搬入ﾌｫｰｸ部在席 1005 / B02から_搬入ﾌｫｰｸ部在席 1005
      MOV     D1453 D346  ; WMＳへ_出庫 搬入 Fork部在席 1005
      DMOV    D3054 D1454  ; B02から_搬入タスクID / B02から_搬入タスクID
      DMOV    D1454 D347  ; WMＳへ_出庫 搬入台 タスクID
      MOV     D3056 D1456  ; B02から_スタッカー受取可 / B02から_スタッカー受取可
      MOV     D1456 D213  ; STKへ_出庫 搬入受取 可
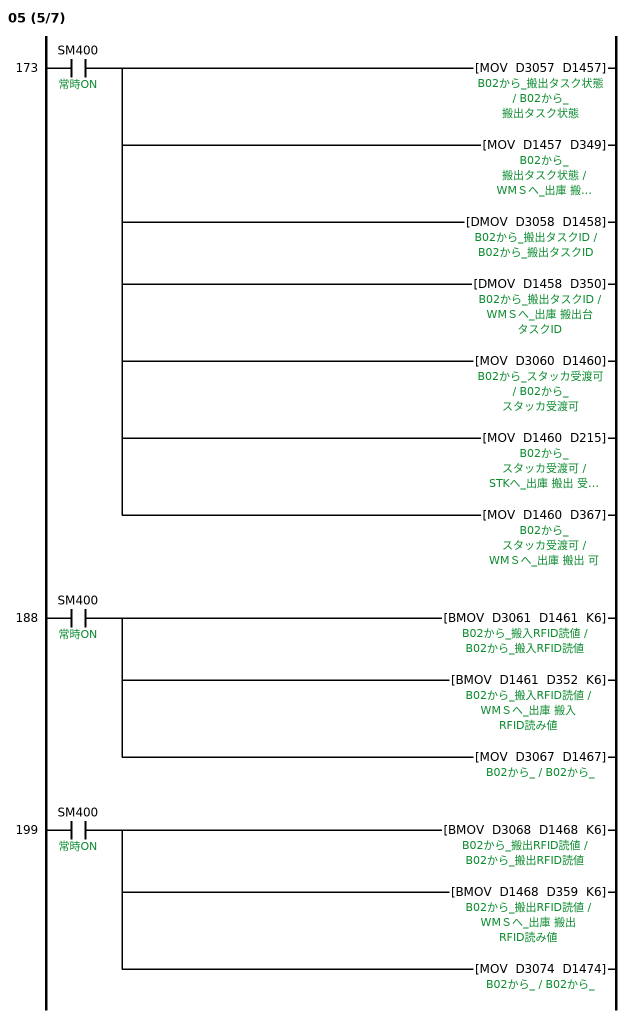
173   LD      SM400  ; 常時ON
      MOV     D3057 D1457  ; B02から_搬出タスク状態 / B02から_搬出タスク状態
      MOV     D1457 D349  ; WMＳへ_出庫 搬出 タスク状態
      DMOV    D3058 D1458  ; B02から_搬出タスクID / B02から_搬出タスクID
      DMOV    D1458 D350  ; WMＳへ_出庫 搬出台 タスクID
      MOV     D3060 D1460  ; B02から_スタッカ受渡可 / B02から_スタッカ受渡可
      MOV     D1460 D215  ; STKへ_出庫 搬出 受渡 可
      MOV     D1460 D367  ; WMＳへ_出庫 搬出 可
188   LD      SM400  ; 常時ON
      BMOV    D3061 D1461 K6  ; B02から_搬入RFID読値 / B02から_搬入RFID読値
      BMOV    D1461 D352 K6  ; WMＳへ_出庫 搬入 RFID読み値
      MOV     D3067 D1467  ; B02から_ / B02から_
199   LD      SM400  ; 常時ON
      BMOV    D3068 D1468 K6  ; B02から_搬出RFID読値 / B02から_搬出RFID読値
      BMOV    D1468 D359 K6  ; WMＳへ_出庫 搬出 RFID読み値
      MOV     D3074 D1474  ; B02から_ / B02から_
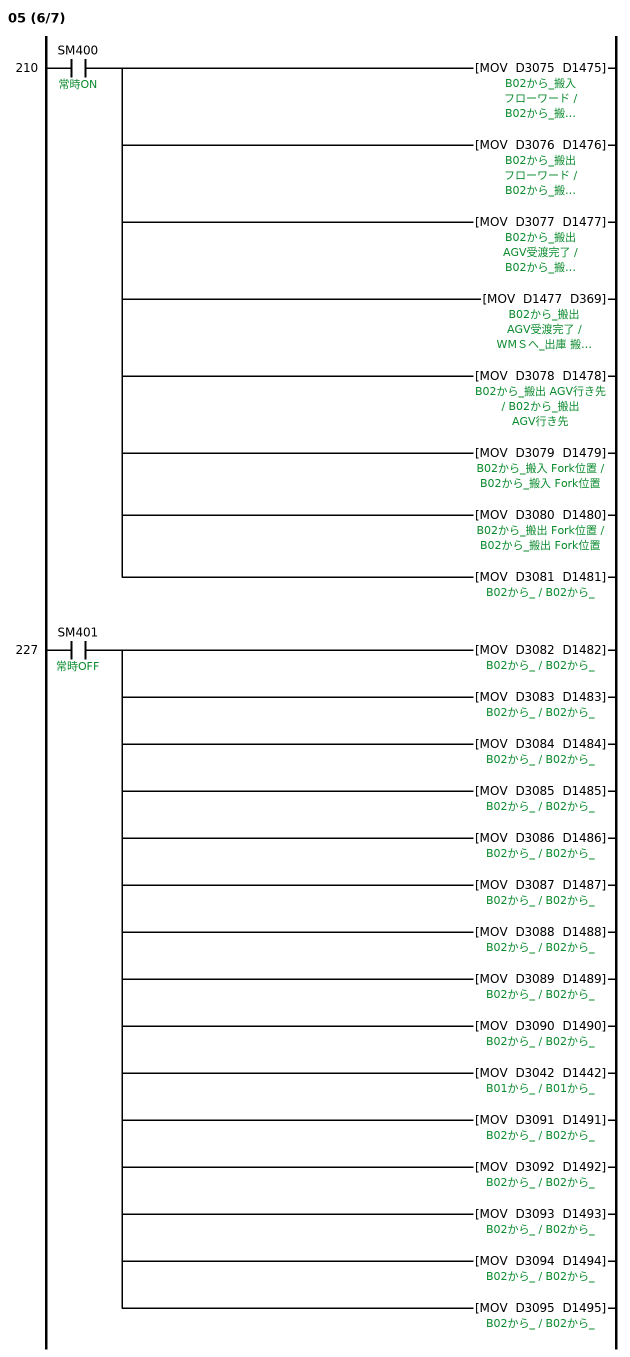
210   LD      SM400  ; 常時ON
      MOV     D3075 D1475  ; B02から_搬入 フローワード / B02から_搬入 フローワード
      MOV     D3076 D1476  ; B02から_搬出 フローワード / B02から_搬出 フローワード
      MOV     D3077 D1477  ; B02から_搬出 AGV受渡完了 / B02から_搬出 AGV受渡完了
      MOV     D1477 D369  ; WMＳへ_出庫 搬出 AGV受渡完了
      MOV     D3078 D1478  ; B02から_搬出 AGV行き先 / B02から_搬出 AGV行き先
      MOV     D3079 D1479  ; B02から_搬入 Fork位置 / B02から_搬入 Fork位置
      MOV     D3080 D1480  ; B02から_搬出 Fork位置 / B02から_搬出 Fork位置
      MOV     D3081 D1481  ; B02から_ / B02から_
227   LD      SM401  ; 常時OFF
      MOV     D3082 D1482  ; B02から_ / B02から_
      MOV     D3083 D1483  ; B02から_ / B02から_
      MOV     D3084 D1484  ; B02から_ / B02から_
      MOV     D3085 D1485  ; B02から_ / B02から_
      MOV     D3086 D1486  ; B02から_ / B02から_
      MOV     D3087 D1487  ; B02から_ / B02から_
      MOV     D3088 D1488  ; B02から_ / B02から_
      MOV     D3089 D1489  ; B02から_ / B02から_
      MOV     D3090 D1490  ; B02から_ / B02から_
      MOV     D3042 D1442  ; B01から_ / B01から_
      MOV     D3091 D1491  ; B02から_ / B02から_
      MOV     D3092 D1492  ; B02から_ / B02から_
      MOV     D3093 D1493  ; B02から_ / B02から_
      MOV     D3094 D1494  ; B02から_ / B02から_
      MOV     D3095 D1495  ; B02から_ / B02から_
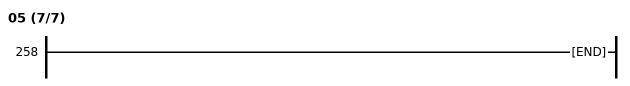
258   END
END_PROGRAM

PROGRAM 45  // B02 CC-LinkIE XVD 出力
0     END
END_PROGRAM

// device comments not shown above
M205  ; HMI_在庫クリアPB
M50  ; XY軸位置決め完了
M207  ; HMi_PC有効PB
M208  ; HMi_PC無効PB
M210  ; HMI_連動PC無効_搬出RFID検索PB
M211  ; HMI_連動PC無効_RFID検索成功
M212  ; HMI_連動PC無効_RFID検索失敗
M219  ; HMI_連動PC無効空き保管庫検索PB
M233  ; HMI_ｽﾀｯｶｰ原点復帰PB
M235  ; HMI PB 手動 位置/棚位置決め
M236  ; HMI PB Y軸強制
M310  ; HMI_STK一時停止PB
M311  ; HMI_STKリセット止PB
M312  ; HMI_STK手動PB要求
M313  ; HMI_ｽﾀｯｶｰ原点復帰PB
M314  ; HMI_STKタスク継続PB
M315  ; HMI_STKタスククリアPB
M360  ; スタッカーSC通信异常
M400  ; STKへ_手動制御リクエスト
M401  ; STKへ__庫位置切替
M402  ; STKへ__Y軸 強制
M403  ; STKへ__X軸 定位
M404  ; STKへ__Y軸 定位
M405  ; STKへ__Z軸 定位
M406  ; STKへ__X軸 前進
M407  ; STKへ__X軸 後退
M408  ; STKへ__Y軸 上昇
M409  ; STKへ__Y軸 下降
M410  ; STKへ__Z軸 左伸
M411  ; STKへ__Z軸 右伸
M412  ; STKへ_原点位置へ動作
M413  ; STKへ_自動運転中
M414  ; STKへ_予備3
M415  ; STKへ_予備4
M1500  ; B01へ_異常リセット
M1501  ; B01へ_受取中
M1502  ; B01へ_受渡中
M1548  ; B02へ_異常リセット
M1549  ; B02へ_受取中
M1550  ; B02へ_受渡中
M2002  ; STKへ__Y軸 強制
M2012  ; STKへ_原点位置へ動作
M2014  ; STKへ_予備3
M2015  ; STKへ_予備4
M2502  ; STKから_前進定位到着
M2503  ; STKから_後退定位到着
M2504  ; STKから_上昇定位到着
M2505  ; STKから_下降定位到着
M2506  ; STKから_左伸定位到着
M2507  ; STKから_右伸定位到着
M2508  ; STKから_受取中
M2509  ; STKから_受渡中
M2510  ; STKから_受取完了
M3214  ; Stacker_Done
M3215  ; パルス
D2  ; GOTｵｰﾊﾞﾗｯﾌﾟｳｨﾝﾄﾞｳ2
D3  ; GOTｵｰﾊﾞﾗｯﾌﾟｳｨﾝﾄﾞｳ3
D4  ; GOTｵｰﾊﾞﾗｯﾌﾟｳｨﾝﾄﾞｳ4
D5  ; GOTｵｰﾊﾞﾗｯﾌﾟｳｨﾝﾄﾞｳ5
D10  ; GOTｼｽﾃﾑ信号1-1
D11  ; GOTｼｽﾃﾑ信号2-1
D13  ; 表示中ｳｨﾝﾄﾞｳ画面1番号
D14  ; 表示中ｳｨﾝﾄﾞｳ画面2番号
D15  ; 表示中ｳｨﾝﾄﾞｳ画面3番号
D16  ; 表示中ｳｨﾝﾄﾞｳ画面4番号
D17  ; 表示中ｳｨﾝﾄﾞｳ画面5番号
D105  ; STKから_現在タスクID
D107  ; STKから_タスク実行総回数
D202  ; STKへ_タスクID
D305  ; WMSへ_現在タスクID
D307  ; WMSへ_タスク実行総回数
D327  ; WMＳへ_入庫 搬入台 タスクID
D330  ; WMＳへ_入庫 搬出台 タスクID
D348  ; WMＳへ_出庫 搬入台 タスクID
D351  ; WMＳへ_出庫 搬出台 タスクID
D402  ; WMSから_タスクID
D451  ; Alarm_  Code
D471  ; 連動_PC無効_搬出口
D502  ; 連動_PC無効_タスクID
D511  ; 連動_PC無効_系统ハートビット
D512  ; 連動_PC無効_入庫 搬入 可
D513  ; 連動_PC無効_出庫 搬入 可
D514  ; 連動_PC無効_入庫 搬出 可
D515  ; 連動_PC無効_出庫 搬出 可
D516  ; 連動_PC無効_アラームリセット
D517  ; 連動_PC無効_予備7
D518  ; 連動_PC無効_予備8
D519  ; 連動_PC無効_予備9
D520  ; 連動_PC無効_予備10
D521  ; 連動_PC無効_入庫 AGV行先
D522  ; 連動_PC無効_出庫 AGV行先
D523  ; 連動_PC無効_入庫 搬入 RFID異常
D524  ; 連動_PC無効_入庫 搬出 RFID異常
D525  ; 連動_PC無効_出庫 搬入 RFID異常
D526  ; 連動_PC無効_出庫 搬出 RFID異常
D527  ; 連動_PC無効_予備17
D528  ; 連動_PC無効_予備18
D529  ; 連動_PC無効_予備19
D1005  ; STKから_現在タスクID
D1007  ; STKから_タスク実行総回数
D1102  ; STKへ_タスクID
D1205  ; WMSへ_現在タスクID
D1207  ; WMSへ_タスク実行総回数
D1227  ; WMＳへ_入庫 搬入台 タスクID
D1230  ; WMＳへ_入庫 搬出台 タスクID
D1248  ; WMＳへ_出庫 搬入台 タスクID
D1251  ; WMＳへ_出庫 搬出台 タスクID
D1302  ; WMSから_タスクID
D1407  ; B01から_搬入タスクID
D1411  ; B01から_搬出タスクID
D1414  ; B01から__搬入RFID読値
D1455  ; B02から_搬入タスクID
D1459  ; B02から_搬出タスクID
D1600  ; B01へ_ ハートビート
D1603  ; B01へ_搬入台 STK受取完了
D1606  ; B01へ_AGVへ出荷許可
D1607  ; B01へ_搬入RFID異常
D1608  ; B01へ_搬出RFID異常
D1611  ; B01へ_地上盤モード現在
D1648  ; B02へ_ ハートビート
D1651  ; B02へ_搬入台 STK受取完了
D1654  ; B02へ_AGVへ出荷許可
D1655  ; B02へ_搬入RFID異常
D1656  ; B02へ_搬出RFID異常
D1659  ; B02へ_地上盤モード現在
D1696  ; AGV統括盤へ_ハートビート
D1697  ; AGV統括盤へ_B01搬出AGV行き先
D1698  ; AGV統括盤へ_B02搬出AGV行き先
D1699  ; AGV統括盤へ_B01搬出AGV発進可
D1700  ; AGV統括盤へ_B02搬出AGV発進可
D3007  ; B01から_搬入タスクID
D3011  ; B01から_搬出タスクID
D3014  ; B01から__搬入RFID読値
D3055  ; B02から_搬入タスクID
D3059  ; B02から_搬出タスクID
D3288  ; Out_CV1.タスクID1
D3290  ; Out_CV1.タスクID2
D3294  ; Out_CV2.タスクID1
D3296  ; Out_CV2.タスクID2
D3300  ; CV2_Out ID
D3302  ; CV1_Out ID
D3303  ; Heartbeat
D4000  ; B01へ_ ハートビート
D4003  ; B01へ_搬入台 STK受取完了
D4011  ; B01へ_地上盤モード現在
D4048  ; B02へ_ ハートビート
D4051  ; B02へ_搬入台 STK受取完了
D4059  ; B02へ_地上盤モード現在
D4096  ; AGV統括盤へ_ハートビート
D4097  ; AGV統括盤へ_B01搬出AGV行き先
D4098  ; AGV統括盤へ_B02搬出AGV行き先
D4099  ; AGV統括盤へ_B01搬出AGV発進可
D4100  ; AGV統括盤へ_B02搬出AGV発進可
Y1000  ; B01へ_異常リセット
Y1001  ; B01へ_受取中
Y1002  ; B01へ_受渡中
Y1030  ; B02へ_異常リセット
Y1031  ; B02へ_受取中
Y1032  ; B02へ_受渡中
B1000  ; 地上→B01_電源 入
B1001  ; 地上→B01_運転準備 入
B1002  ; 地上→B01_重故障
B1003  ; 地上→B01_軽故障
B1004  ; 地上→B01_非常停止 正常
B100A  ; 地上→B01_自動運転中
B100B  ; 地上→B01_サイクル停止中
B100C  ; 地上→B01_手動操作中
B100D  ; 地上→B01_特殊操作中
B1010  ; 地上→B01_自動モード選択
B1011  ; 地上→B01_手動モード選択
B1012  ; 地上→B01_連動モード選択
B1013  ; 地上→B01_単独モード選択
B1014  ; 地上→B01_管理者モード選択
B101A  ; 地上→B01_連動 起動
B101B  ; 地上→B01_連動 サイクル停止
B1020  ; 地上→B01_入庫側 搬入 受取中
B1021  ; 地上→B01_入庫側 搬入 受取完了
B1022  ; 地上→B01_入庫側 搬出 受渡中
B1023  ; 地上→B01_入庫側 搬出 受渡完了
B102A  ; 地上→B01_入庫側 搬入 RFID 再取
B102B  ; 地上→B01_入庫側 搬出 RFID 再取
B1100  ; 地上→B02_電源 入
B1101  ; 地上→B02_運転準備 入
B1102  ; 地上→B02_重故障
B1103  ; 地上→B02_軽故障
B1104  ; 地上→B02_非常停止 正常
B110A  ; 地上→B02_自動運転中
B110B  ; 地上→B02_サイクル停止中
B110C  ; 地上→B02_手動操作中
B110D  ; 地上→B02_特殊操作中
B1110  ; 地上→B02_自動モード選択
B1111  ; 地上→B02_手動モード選択
B1112  ; 地上→B02_連動モード選択
B1113  ; 地上→B02_単独モード選択
B1114  ; 地上→B02_管理者モード選択
B1115  ; 地上→B02予備
B1117  ; 地上→B03予備
B1118  ; 地上→B03_予備
B1119  ; 地上→B04予備
B111A  ; 地上→_連動 起動
B111B  ; 地上→_連動 サイクル停止
B1120  ; 地上→B02_出庫側 搬入 受取中
B1121  ; 地上→B02_出庫側 搬入 受取完了
B1122  ; 地上→B02_出庫側 搬出 受取中
B1123  ; 地上→B02_出庫側 搬出 受取完了
B112A  ; 地上→B02_出庫側 搬入 RFID 再取
B112B  ; 地上→B02_出庫側 搬出 RFID 再取
W900.0  ; ステション 1
